// Block: PTrk_HMI

DATA_BLOCK PTrk_HMI
VERSION : 0.1
   NON_RETAIN
   VAR
      Button_Part_Recondition_Good : Struct
         Show : Bool;
         AllowControl : Bool;
         Pressed : Bool;
      END_STRUCT;
      Button_Part_Recondition_NG : Struct
         Show : Bool;
         AllowControl : Bool;
         Pressed : Bool;
      END_STRUCT;
   END_VAR

BEGIN
   // No initialization required
END_DATA_BLOCK
